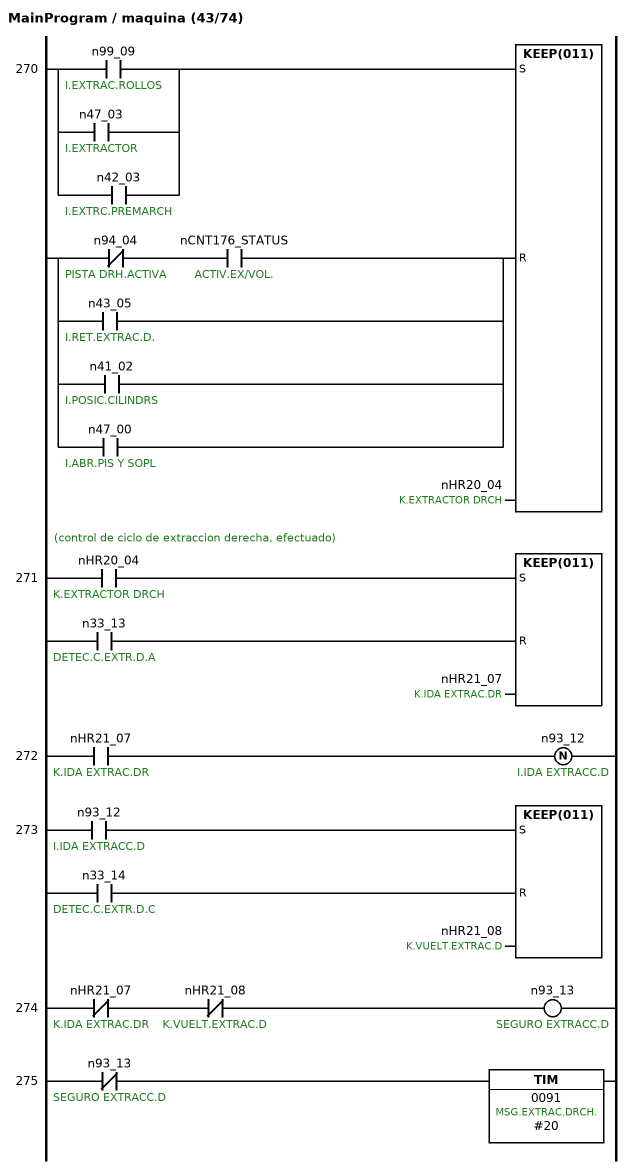
; [picture p48: MainProgram / maquina, rungs 270-275]
; rung 270
LD n99_09  ; I.EXTRAC.ROLLOS
OR n47_03  ; I.EXTRACTOR
OR n42_03  ; I.EXTRC.PREMARCH
LDNOT n94_04  ; PISTA DRH.ACTIVA
AND nCNT176_STATUS  ; ACTIV.EX/VOL.
OR n43_05  ; I.RET.EXTRAC.D.
OR n41_02  ; I.POSIC.CILINDRS
OR n47_00  ; I.ABR.PIS Y SOPL
KEEP(011) nHR20_04  ; K.EXTRACTOR DRCH
; rung 271: (control de ciclo de extraccion derecha, efectuado)
LD nHR20_04  ; K.EXTRACTOR DRCH
LD n33_13  ; DETEC.C.EXTR.D.A
KEEP(011) nHR21_07  ; K.IDA EXTRAC.DR
; rung 272
LD nHR21_07  ; K.IDA EXTRAC.DR
DIFD(014) n93_12  ; I.IDA EXTRACC.D
; rung 273
LD n93_12  ; I.IDA EXTRACC.D
LD n33_14  ; DETEC.C.EXTR.D.C
KEEP(011) nHR21_08  ; K.VUELT.EXTRAC.D
; rung 274
LDNOT nHR21_07  ; K.IDA EXTRAC.DR
ANDNOT nHR21_08  ; K.VUELT.EXTRAC.D
OUT n93_13  ; SEGURO EXTRACC.D
; rung 275
LDNOT n93_13  ; SEGURO EXTRACC.D
TIM 0091 #20  ; MSG.EXTRAC.DRCH.

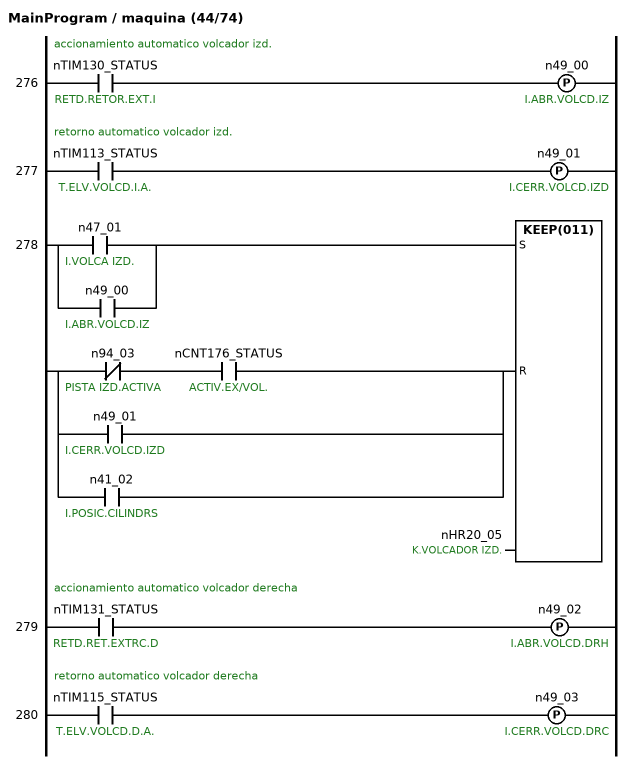
; rung 276: accionamiento automatico volcador izd.
LD nTIM130_STATUS  ; RETD.RETOR.EXT.I
DIFU(013) n49_00  ; I.ABR.VOLCD.IZ
; rung 277: retorno automatico volcador izd.
LD nTIM113_STATUS  ; T.ELV.VOLCD.I.A.
DIFU(013) n49_01  ; I.CERR.VOLCD.IZD
; rung 278
LD n47_01  ; I.VOLCA IZD.
OR n49_00  ; I.ABR.VOLCD.IZ
LDNOT n94_03  ; PISTA IZD.ACTIVA
AND nCNT176_STATUS  ; ACTIV.EX/VOL.
OR n49_01  ; I.CERR.VOLCD.IZD
OR n41_02  ; I.POSIC.CILINDRS
KEEP(011) nHR20_05  ; K.VOLCADOR IZD.
; rung 279: accionamiento automatico volcador derecha
LD nTIM131_STATUS  ; RETD.RET.EXTRC.D
DIFU(013) n49_02  ; I.ABR.VOLCD.DRH
; rung 280: retorno automatico volcador derecha
LD nTIM115_STATUS  ; T.ELV.VOLCD.D.A.
DIFU(013) n49_03  ; I.CERR.VOLCD.DRC

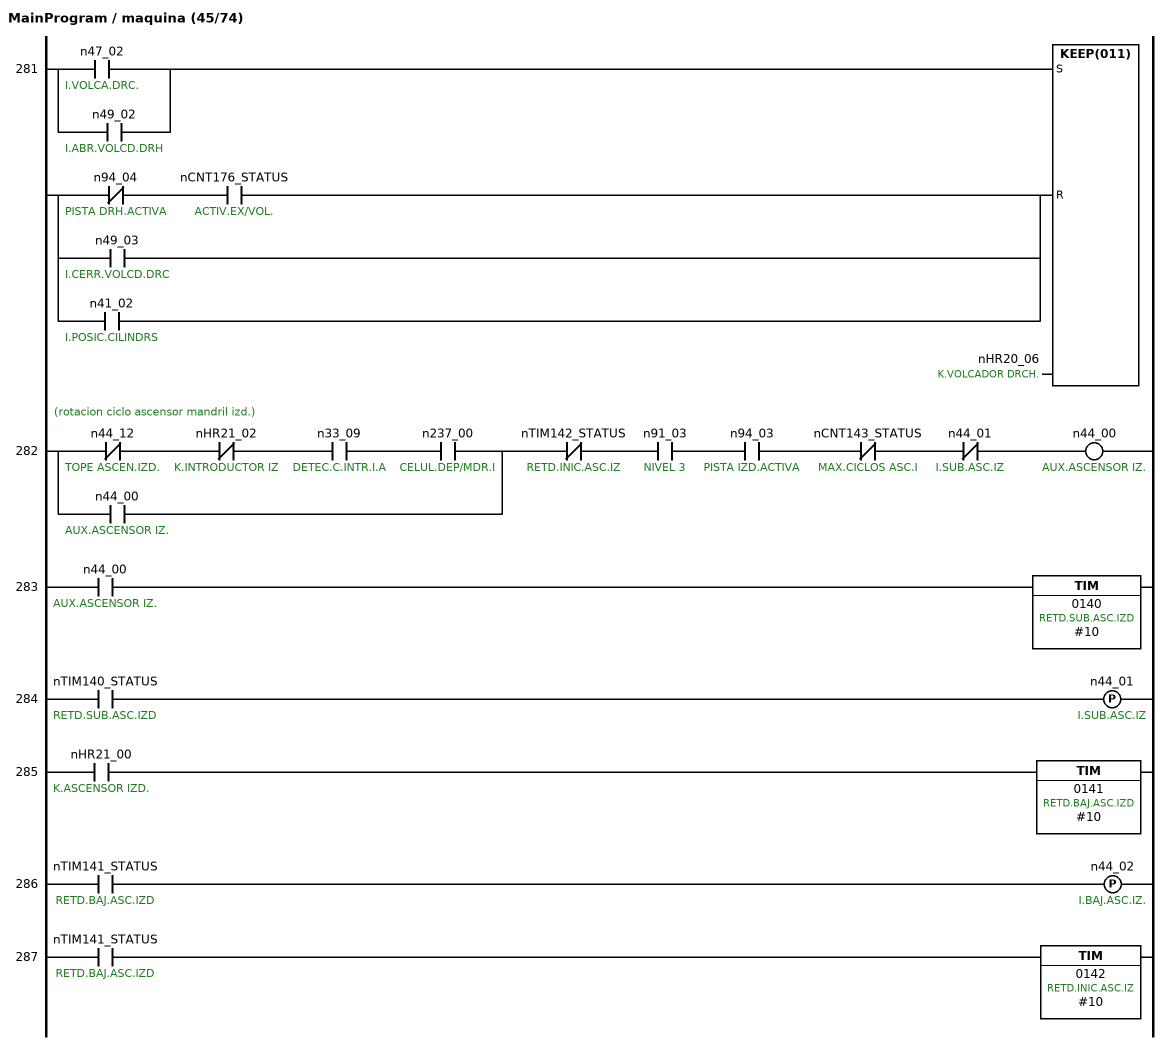
; rung 281
LD n47_02  ; I.VOLCA.DRC.
OR n49_02  ; I.ABR.VOLCD.DRH
LDNOT n94_04  ; PISTA DRH.ACTIVA
AND nCNT176_STATUS  ; ACTIV.EX/VOL.
OR n49_03  ; I.CERR.VOLCD.DRC
OR n41_02  ; I.POSIC.CILINDRS
KEEP(011) nHR20_06  ; K.VOLCADOR DRCH.
; rung 282: (rotacion ciclo ascensor mandril izd.)
LDNOT n44_12  ; TOPE ASCEN.IZD.
ANDNOT nHR21_02  ; K.INTRODUCTOR IZ
AND n33_09  ; DETEC.C.INTR.I.A
AND n237_00  ; CELUL.DEP/MDR.I
OR n44_00  ; AUX.ASCENSOR IZ.
ANDNOT nTIM142_STATUS  ; RETD.INIC.ASC.IZ
AND n91_03  ; NIVEL 3
AND n94_03  ; PISTA IZD.ACTIVA
ANDNOT nCNT143_STATUS  ; MAX.CICLOS ASC.I
ANDNOT n44_01  ; I.SUB.ASC.IZ
OUT n44_00  ; AUX.ASCENSOR IZ.
; rung 283
LD n44_00  ; AUX.ASCENSOR IZ.
TIM 0140 #10  ; RETD.SUB.ASC.IZD
; rung 284
LD nTIM140_STATUS  ; RETD.SUB.ASC.IZD
DIFU(013) n44_01  ; I.SUB.ASC.IZ
; rung 285
LD nHR21_00  ; K.ASCENSOR IZD.
TIM 0141 #10  ; RETD.BAJ.ASC.IZD
; rung 286
LD nTIM141_STATUS  ; RETD.BAJ.ASC.IZD
DIFU(013) n44_02  ; I.BAJ.ASC.IZ.
; rung 287
LD nTIM141_STATUS  ; RETD.BAJ.ASC.IZD
TIM 0142 #10  ; RETD.INIC.ASC.IZ

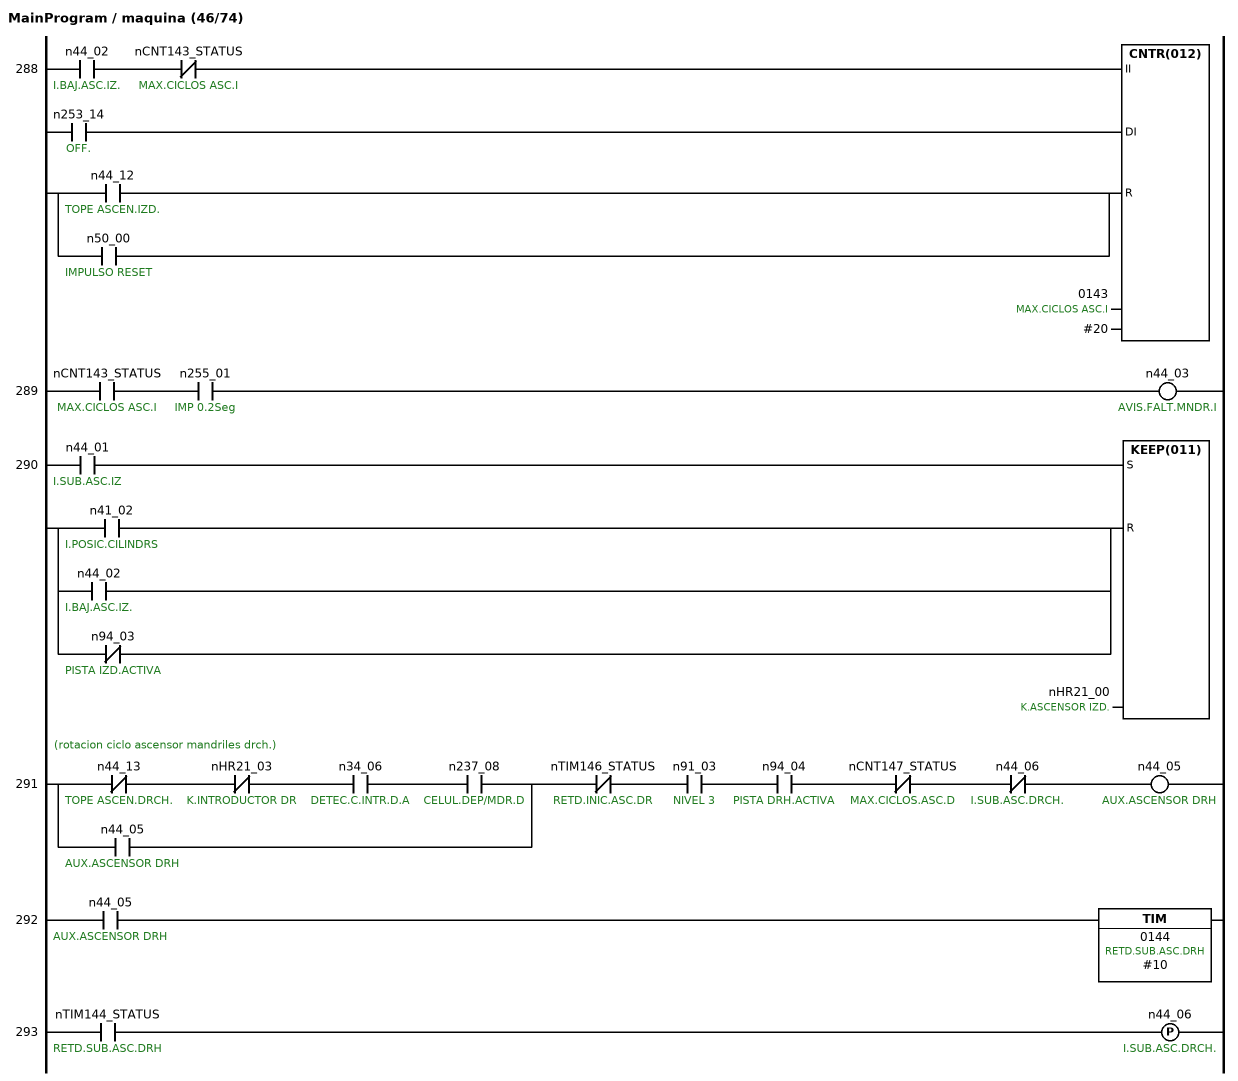
; rung 288
LD n44_02  ; I.BAJ.ASC.IZ.
ANDNOT nCNT143_STATUS  ; MAX.CICLOS ASC.I
LD n253_14  ; OFF.
LD n44_12  ; TOPE ASCEN.IZD.
OR n50_00  ; IMPULSO RESET
CNTR(012) 0143 #20  ; MAX.CICLOS ASC.I
; rung 289
LD nCNT143_STATUS  ; MAX.CICLOS ASC.I
AND n255_01  ; IMP 0.2Seg
OUT n44_03  ; AVIS.FALT.MNDR.I
; rung 290
LD n44_01  ; I.SUB.ASC.IZ
LD n41_02  ; I.POSIC.CILINDRS
OR n44_02  ; I.BAJ.ASC.IZ.
ORNOT n94_03  ; PISTA IZD.ACTIVA
KEEP(011) nHR21_00  ; K.ASCENSOR IZD.
; rung 291: (rotacion ciclo ascensor mandriles drch.)
LDNOT n44_13  ; TOPE ASCEN.DRCH.
ANDNOT nHR21_03  ; K.INTRODUCTOR DR
AND n34_06  ; DETEC.C.INTR.D.A
AND n237_08  ; CELUL.DEP/MDR.D
OR n44_05  ; AUX.ASCENSOR DRH
ANDNOT nTIM146_STATUS  ; RETD.INIC.ASC.DR
AND n91_03  ; NIVEL 3
AND n94_04  ; PISTA DRH.ACTIVA
ANDNOT nCNT147_STATUS  ; MAX.CICLOS.ASC.D
ANDNOT n44_06  ; I.SUB.ASC.DRCH.
OUT n44_05  ; AUX.ASCENSOR DRH
; rung 292
LD n44_05  ; AUX.ASCENSOR DRH
TIM 0144 #10  ; RETD.SUB.ASC.DRH
; rung 293
LD nTIM144_STATUS  ; RETD.SUB.ASC.DRH
DIFU(013) n44_06  ; I.SUB.ASC.DRCH.

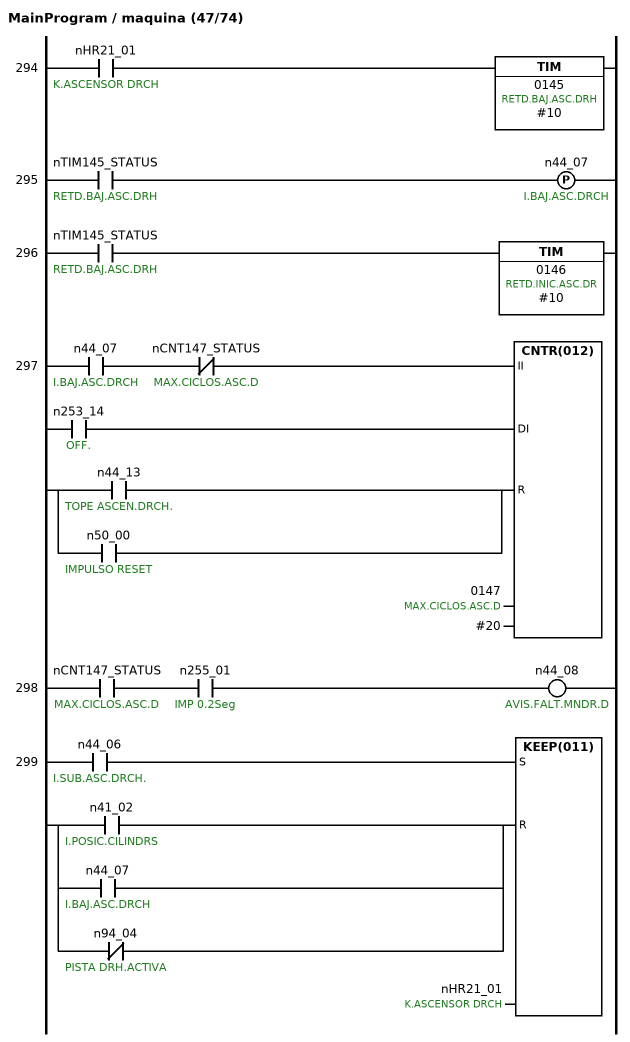
; rung 294
LD nHR21_01  ; K.ASCENSOR DRCH
TIM 0145 #10  ; RETD.BAJ.ASC.DRH
; rung 295
LD nTIM145_STATUS  ; RETD.BAJ.ASC.DRH
DIFU(013) n44_07  ; I.BAJ.ASC.DRCH
; rung 296
LD nTIM145_STATUS  ; RETD.BAJ.ASC.DRH
TIM 0146 #10  ; RETD.INIC.ASC.DR
; rung 297
LD n44_07  ; I.BAJ.ASC.DRCH
ANDNOT nCNT147_STATUS  ; MAX.CICLOS.ASC.D
LD n253_14  ; OFF.
LD n44_13  ; TOPE ASCEN.DRCH.
OR n50_00  ; IMPULSO RESET
CNTR(012) 0147 #20  ; MAX.CICLOS.ASC.D
; rung 298
LD nCNT147_STATUS  ; MAX.CICLOS.ASC.D
AND n255_01  ; IMP 0.2Seg
OUT n44_08  ; AVIS.FALT.MNDR.D
; rung 299
LD n44_06  ; I.SUB.ASC.DRCH.
LD n41_02  ; I.POSIC.CILINDRS
OR n44_07  ; I.BAJ.ASC.DRCH
ORNOT n94_04  ; PISTA DRH.ACTIVA
KEEP(011) nHR21_01  ; K.ASCENSOR DRCH

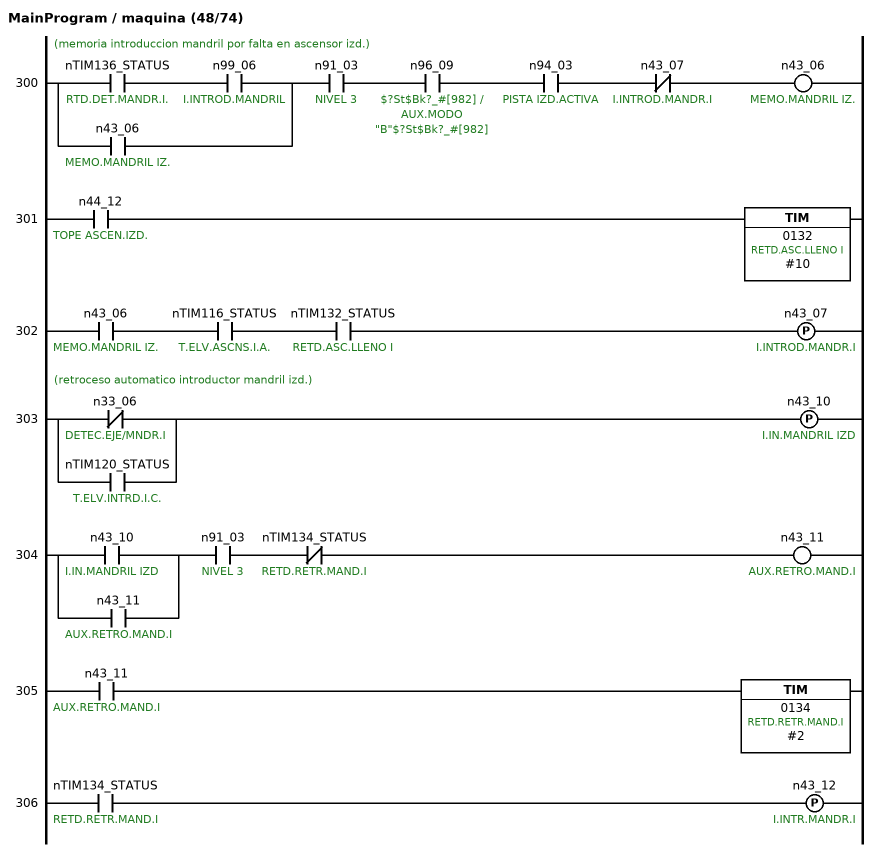
; rung 300: (memoria introduccion mandril por falta en ascensor izd.)
LD nTIM136_STATUS  ; RTD.DET.MANDR.I.
AND n99_06  ; I.INTROD.MANDRIL
OR n43_06  ; MEMO.MANDRIL IZ.
AND n91_03  ; NIVEL 3
AND n96_09  ; $?St$Bk?_#[982] / AUX.MODO "B"$?St$Bk?_#[982]
AND n94_03  ; PISTA IZD.ACTIVA
ANDNOT n43_07  ; I.INTROD.MANDR.I
OUT n43_06  ; MEMO.MANDRIL IZ.
; rung 301
LD n44_12  ; TOPE ASCEN.IZD.
TIM 0132 #10  ; RETD.ASC.LLENO I
; rung 302
LD n43_06  ; MEMO.MANDRIL IZ.
AND nTIM116_STATUS  ; T.ELV.ASCNS.I.A.
AND nTIM132_STATUS  ; RETD.ASC.LLENO I
DIFU(013) n43_07  ; I.INTROD.MANDR.I
; rung 303: (retroceso automatico introductor mandril izd.)
LDNOT n33_06  ; DETEC.EJE/MNDR.I
OR nTIM120_STATUS  ; T.ELV.INTRD.I.C.
DIFU(013) n43_10  ; I.IN.MANDRIL IZD
; rung 304
LD n43_10  ; I.IN.MANDRIL IZD
OR n43_11  ; AUX.RETRO.MAND.I
AND n91_03  ; NIVEL 3
ANDNOT nTIM134_STATUS  ; RETD.RETR.MAND.I
OUT n43_11  ; AUX.RETRO.MAND.I
; rung 305
LD n43_11  ; AUX.RETRO.MAND.I
TIM 0134 #2  ; RETD.RETR.MAND.I
; rung 306
LD nTIM134_STATUS  ; RETD.RETR.MAND.I
DIFU(013) n43_12  ; I.INTR.MANDR.I

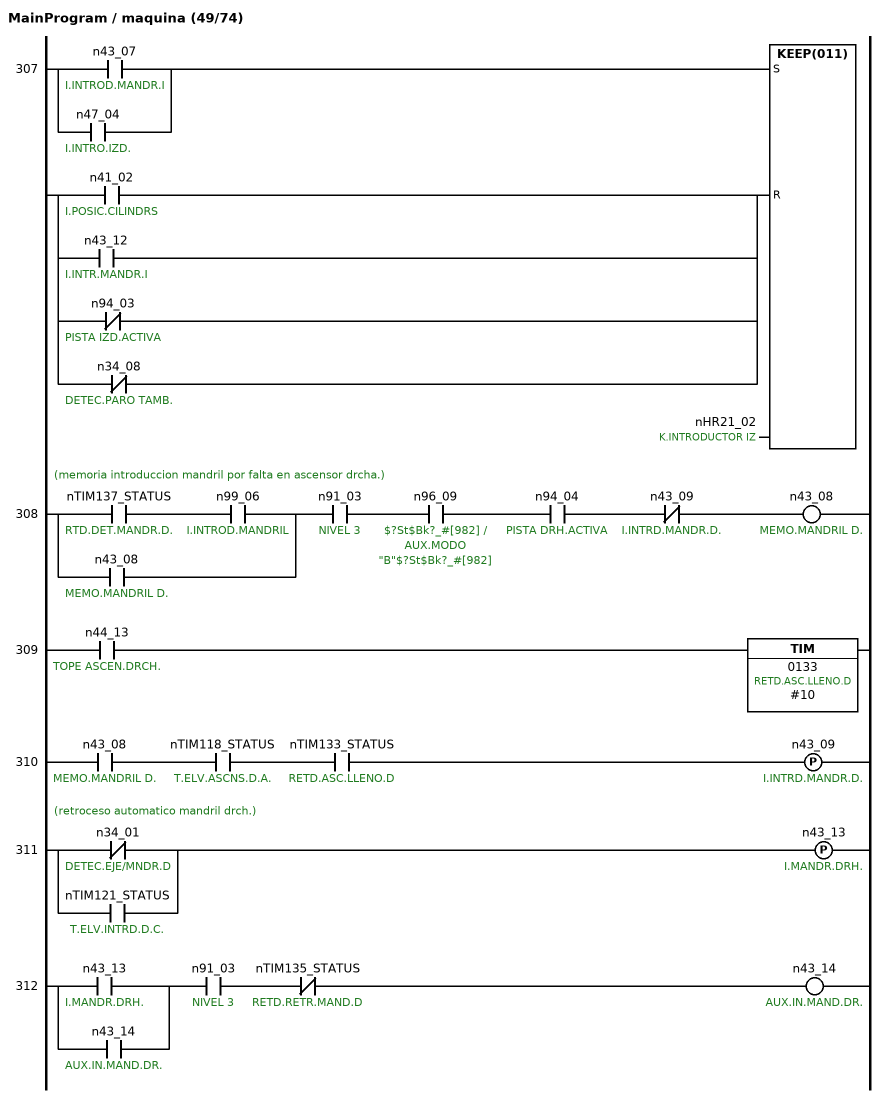
; rung 307
LD n43_07  ; I.INTROD.MANDR.I
OR n47_04  ; I.INTRO.IZD.
LD n41_02  ; I.POSIC.CILINDRS
OR n43_12  ; I.INTR.MANDR.I
ORNOT n94_03  ; PISTA IZD.ACTIVA
ORNOT n34_08  ; DETEC.PARO TAMB.
KEEP(011) nHR21_02  ; K.INTRODUCTOR IZ
; rung 308: (memoria introduccion mandril por falta en ascensor drcha.)
LD nTIM137_STATUS  ; RTD.DET.MANDR.D.
AND n99_06  ; I.INTROD.MANDRIL
OR n43_08  ; MEMO.MANDRIL D.
AND n91_03  ; NIVEL 3
AND n96_09  ; $?St$Bk?_#[982] / AUX.MODO "B"$?St$Bk?_#[982]
AND n94_04  ; PISTA DRH.ACTIVA
ANDNOT n43_09  ; I.INTRD.MANDR.D.
OUT n43_08  ; MEMO.MANDRIL D.
; rung 309
LD n44_13  ; TOPE ASCEN.DRCH.
TIM 0133 #10  ; RETD.ASC.LLENO.D
; rung 310
LD n43_08  ; MEMO.MANDRIL D.
AND nTIM118_STATUS  ; T.ELV.ASCNS.D.A.
AND nTIM133_STATUS  ; RETD.ASC.LLENO.D
DIFU(013) n43_09  ; I.INTRD.MANDR.D.
; rung 311: (retroceso automatico mandril drch.)
LDNOT n34_01  ; DETEC.EJE/MNDR.D
OR nTIM121_STATUS  ; T.ELV.INTRD.D.C.
DIFU(013) n43_13  ; I.MANDR.DRH.
; rung 312
LD n43_13  ; I.MANDR.DRH.
OR n43_14  ; AUX.IN.MAND.DR.
AND n91_03  ; NIVEL 3
ANDNOT nTIM135_STATUS  ; RETD.RETR.MAND.D
OUT n43_14  ; AUX.IN.MAND.DR.

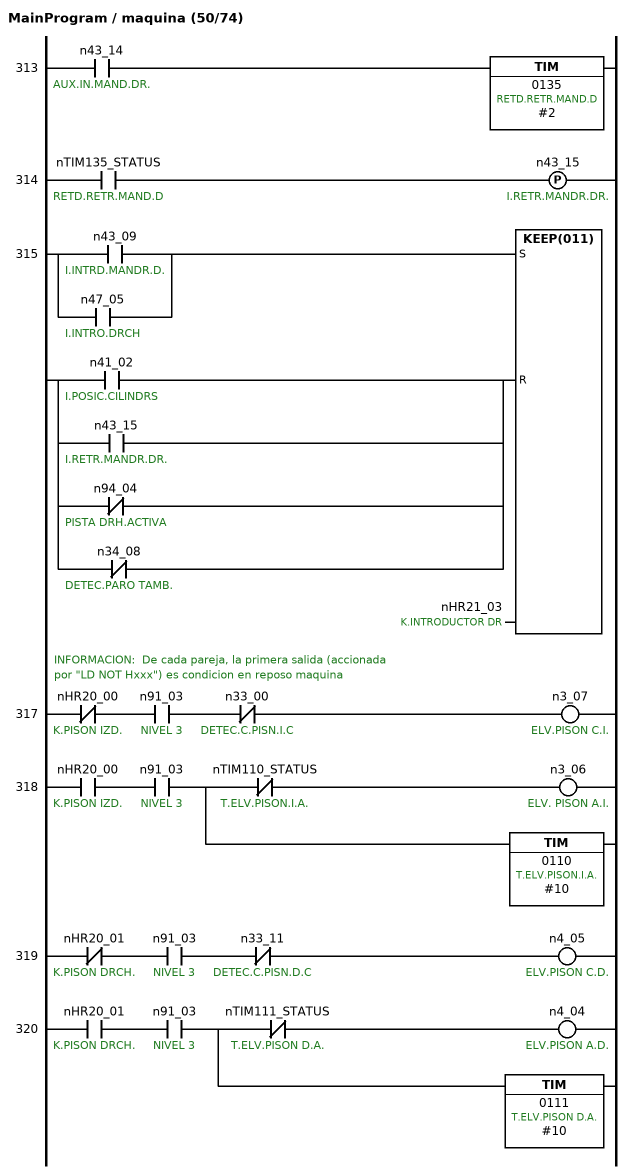
; rung 313
LD n43_14  ; AUX.IN.MAND.DR.
TIM 0135 #2  ; RETD.RETR.MAND.D
; rung 314
LD nTIM135_STATUS  ; RETD.RETR.MAND.D
DIFU(013) n43_15  ; I.RETR.MANDR.DR.
; rung 315
LD n43_09  ; I.INTRD.MANDR.D.
OR n47_05  ; I.INTRO.DRCH
LD n41_02  ; I.POSIC.CILINDRS
OR n43_15  ; I.RETR.MANDR.DR.
ORNOT n94_04  ; PISTA DRH.ACTIVA
ORNOT n34_08  ; DETEC.PARO TAMB.
KEEP(011) nHR21_03  ; K.INTRODUCTOR DR
; rung 316: ACCIONAMIENTO ELVS. REBOBINADOR, VOLCADORES Y CARGADORES / ------------------------------------------------------------
; rung 317: INFORMACION:  De cada pareja, la primera salida (accionada / por "LD NOT Hxxx") es condicion en reposo maquina
LDNOT nHR20_00  ; K.PISON IZD.
AND n91_03  ; NIVEL 3
ANDNOT n33_00  ; DETEC.C.PISN.I.C
OUT n3_07  ; ELV.PISON C.I.
; rung 318
LD nHR20_00  ; K.PISON IZD.
AND n91_03  ; NIVEL 3
OUT TR0
ANDNOT nTIM110_STATUS  ; T.ELV.PISON.I.A.
OUT n3_06  ; ELV. PISON A.I.
LD TR0
TIM 0110 #10  ; T.ELV.PISON.I.A.
; rung 319
LDNOT nHR20_01  ; K.PISON DRCH.
AND n91_03  ; NIVEL 3
ANDNOT n33_11  ; DETEC.C.PISN.D.C
OUT n4_05  ; ELV.PISON C.D.
; rung 320
LD nHR20_01  ; K.PISON DRCH.
AND n91_03  ; NIVEL 3
OUT TR0
ANDNOT nTIM111_STATUS  ; T.ELV.PISON D.A.
OUT n4_04  ; ELV.PISON A.D.
LD TR0
TIM 0111 #10  ; T.ELV.PISON D.A.

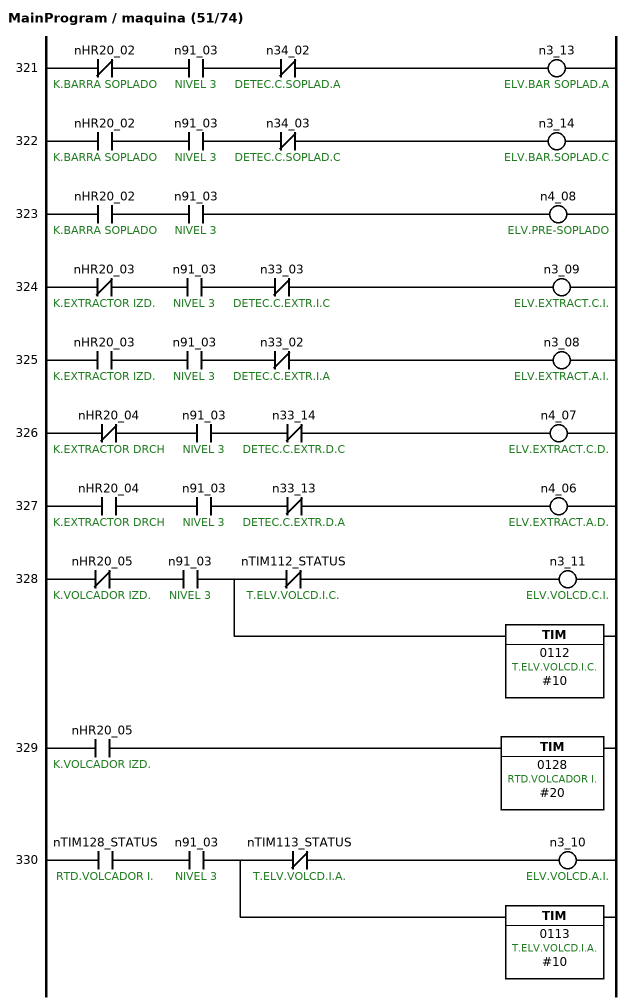
; rung 321
LDNOT nHR20_02  ; K.BARRA SOPLADO
AND n91_03  ; NIVEL 3
ANDNOT n34_02  ; DETEC.C.SOPLAD.A
OUT n3_13  ; ELV.BAR SOPLAD.A
; rung 322
LD nHR20_02  ; K.BARRA SOPLADO
AND n91_03  ; NIVEL 3
ANDNOT n34_03  ; DETEC.C.SOPLAD.C
OUT n3_14  ; ELV.BAR.SOPLAD.C
; rung 323
LD nHR20_02  ; K.BARRA SOPLADO
AND n91_03  ; NIVEL 3
OUT n4_08  ; ELV.PRE-SOPLADO
; rung 324
LDNOT nHR20_03  ; K.EXTRACTOR IZD.
AND n91_03  ; NIVEL 3
ANDNOT n33_03  ; DETEC.C.EXTR.I.C
OUT n3_09  ; ELV.EXTRACT.C.I.
; rung 325
LD nHR20_03  ; K.EXTRACTOR IZD.
AND n91_03  ; NIVEL 3
ANDNOT n33_02  ; DETEC.C.EXTR.I.A
OUT n3_08  ; ELV.EXTRACT.A.I.
; rung 326
LDNOT nHR20_04  ; K.EXTRACTOR DRCH
AND n91_03  ; NIVEL 3
ANDNOT n33_14  ; DETEC.C.EXTR.D.C
OUT n4_07  ; ELV.EXTRACT.C.D.
; rung 327
LD nHR20_04  ; K.EXTRACTOR DRCH
AND n91_03  ; NIVEL 3
ANDNOT n33_13  ; DETEC.C.EXTR.D.A
OUT n4_06  ; ELV.EXTRACT.A.D.
; rung 328
LDNOT nHR20_05  ; K.VOLCADOR IZD.
AND n91_03  ; NIVEL 3
OUT TR0
ANDNOT nTIM112_STATUS  ; T.ELV.VOLCD.I.C.
OUT n3_11  ; ELV.VOLCD.C.I.
LD TR0
TIM 0112 #10  ; T.ELV.VOLCD.I.C.
; rung 329
LD nHR20_05  ; K.VOLCADOR IZD.
TIM 0128 #20  ; RTD.VOLCADOR I.
; rung 330
LD nTIM128_STATUS  ; RTD.VOLCADOR I.
AND n91_03  ; NIVEL 3
OUT TR0
ANDNOT nTIM113_STATUS  ; T.ELV.VOLCD.I.A.
OUT n3_10  ; ELV.VOLCD.A.I.
LD TR0
TIM 0113 #10  ; T.ELV.VOLCD.I.A.

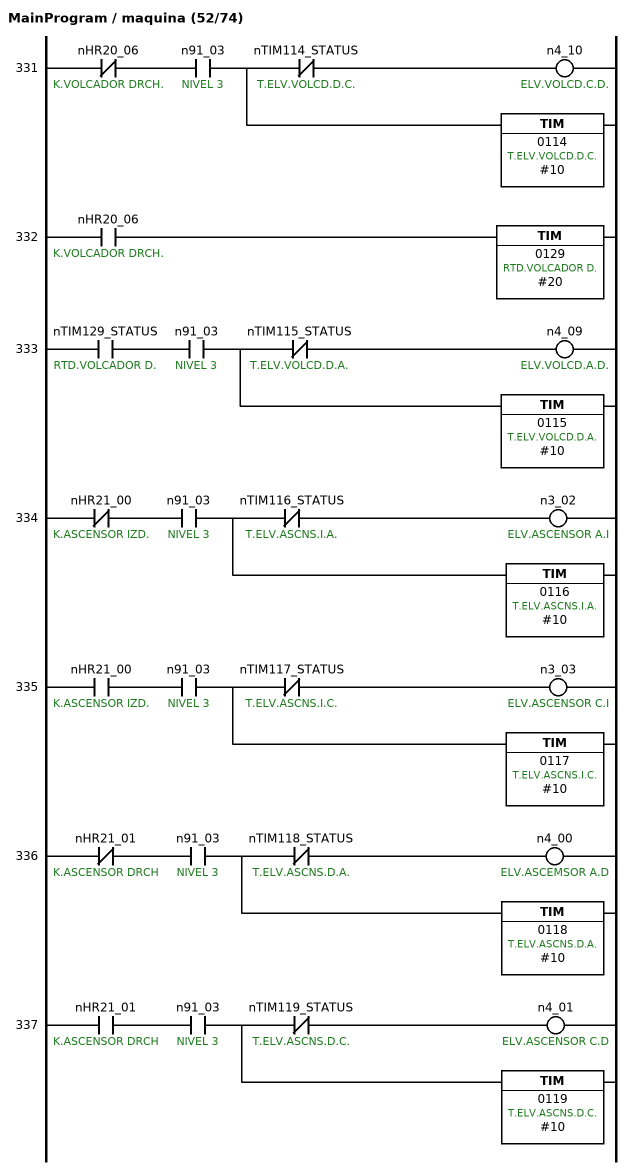
; rung 331
LDNOT nHR20_06  ; K.VOLCADOR DRCH.
AND n91_03  ; NIVEL 3
OUT TR0
ANDNOT nTIM114_STATUS  ; T.ELV.VOLCD.D.C.
OUT n4_10  ; ELV.VOLCD.C.D.
LD TR0
TIM 0114 #10  ; T.ELV.VOLCD.D.C.
; rung 332
LD nHR20_06  ; K.VOLCADOR DRCH.
TIM 0129 #20  ; RTD.VOLCADOR D.
; rung 333
LD nTIM129_STATUS  ; RTD.VOLCADOR D.
AND n91_03  ; NIVEL 3
OUT TR0
ANDNOT nTIM115_STATUS  ; T.ELV.VOLCD.D.A.
OUT n4_09  ; ELV.VOLCD.A.D.
LD TR0
TIM 0115 #10  ; T.ELV.VOLCD.D.A.
; rung 334
LDNOT nHR21_00  ; K.ASCENSOR IZD.
AND n91_03  ; NIVEL 3
OUT TR0
ANDNOT nTIM116_STATUS  ; T.ELV.ASCNS.I.A.
OUT n3_02  ; ELV.ASCENSOR A.I
LD TR0
TIM 0116 #10  ; T.ELV.ASCNS.I.A.
; rung 335
LD nHR21_00  ; K.ASCENSOR IZD.
AND n91_03  ; NIVEL 3
OUT TR0
ANDNOT nTIM117_STATUS  ; T.ELV.ASCNS.I.C.
OUT n3_03  ; ELV.ASCENSOR C.I
LD TR0
TIM 0117 #10  ; T.ELV.ASCNS.I.C.
; rung 336
LDNOT nHR21_01  ; K.ASCENSOR DRCH
AND n91_03  ; NIVEL 3
OUT TR0
ANDNOT nTIM118_STATUS  ; T.ELV.ASCNS.D.A.
OUT n4_00  ; ELV.ASCEMSOR A.D
LD TR0
TIM 0118 #10  ; T.ELV.ASCNS.D.A.
; rung 337
LD nHR21_01  ; K.ASCENSOR DRCH
AND n91_03  ; NIVEL 3
OUT TR0
ANDNOT nTIM119_STATUS  ; T.ELV.ASCNS.D.C.
OUT n4_01  ; ELV.ASCENSOR C.D
LD TR0
TIM 0119 #10  ; T.ELV.ASCNS.D.C.

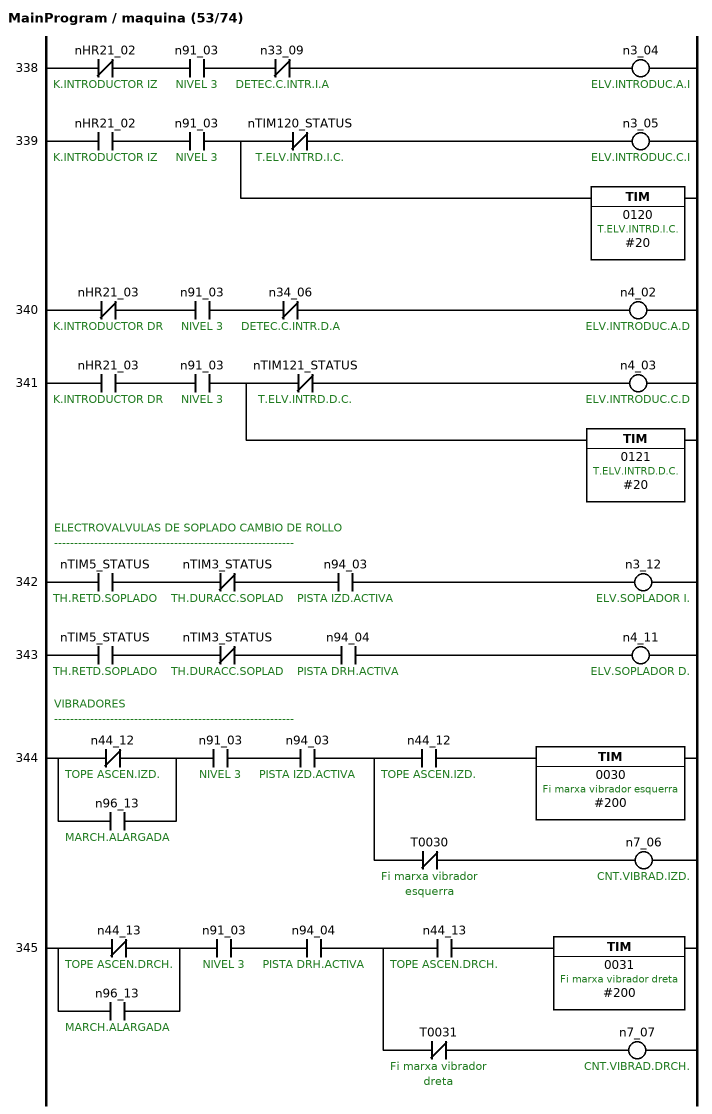
; rung 338
LDNOT nHR21_02  ; K.INTRODUCTOR IZ
AND n91_03  ; NIVEL 3
ANDNOT n33_09  ; DETEC.C.INTR.I.A
OUT n3_04  ; ELV.INTRODUC.A.I
; rung 339
LD nHR21_02  ; K.INTRODUCTOR IZ
AND n91_03  ; NIVEL 3
OUT TR0
ANDNOT nTIM120_STATUS  ; T.ELV.INTRD.I.C.
OUT n3_05  ; ELV.INTRODUC.C.I
LD TR0
TIM 0120 #20  ; T.ELV.INTRD.I.C.
; rung 340
LDNOT nHR21_03  ; K.INTRODUCTOR DR
AND n91_03  ; NIVEL 3
ANDNOT n34_06  ; DETEC.C.INTR.D.A
OUT n4_02  ; ELV.INTRODUC.A.D
; rung 341
LD nHR21_03  ; K.INTRODUCTOR DR
AND n91_03  ; NIVEL 3
OUT TR0
ANDNOT nTIM121_STATUS  ; T.ELV.INTRD.D.C.
OUT n4_03  ; ELV.INTRODUC.C.D
LD TR0
TIM 0121 #20  ; T.ELV.INTRD.D.C.
; rung 342: ELECTROVALVULAS DE SOPLADO CAMBIO DE ROLLO / ------------------------------------------------------------
LD nTIM5_STATUS  ; TH.RETD.SOPLADO
ANDNOT nTIM3_STATUS  ; TH.DURACC.SOPLAD
AND n94_03  ; PISTA IZD.ACTIVA
OUT n3_12  ; ELV.SOPLADOR I.
; rung 343
LD nTIM5_STATUS  ; TH.RETD.SOPLADO
ANDNOT nTIM3_STATUS  ; TH.DURACC.SOPLAD
AND n94_04  ; PISTA DRH.ACTIVA
OUT n4_11  ; ELV.SOPLADOR D.
; rung 344: VIBRADORES / ------------------------------------------------------------
LDNOT n44_12  ; TOPE ASCEN.IZD.
OR n96_13  ; MARCH.ALARGADA
AND n91_03  ; NIVEL 3
AND n94_03  ; PISTA IZD.ACTIVA
OUT TR0
AND n44_12  ; TOPE ASCEN.IZD.
TIM 0030 #200  ; Fi marxa vibrador esquerra
LD TR0
ANDNOT T0030  ; Fi marxa vibrador esquerra
OUT n7_06  ; CNT.VIBRAD.IZD.
; rung 345
LDNOT n44_13  ; TOPE ASCEN.DRCH.
OR n96_13  ; MARCH.ALARGADA
AND n91_03  ; NIVEL 3
AND n94_04  ; PISTA DRH.ACTIVA
OUT TR0
AND n44_13  ; TOPE ASCEN.DRCH.
TIM 0031 #200  ; Fi marxa vibrador dreta
LD TR0
ANDNOT T0031  ; Fi marxa vibrador dreta
OUT n7_07  ; CNT.VIBRAD.DRCH.

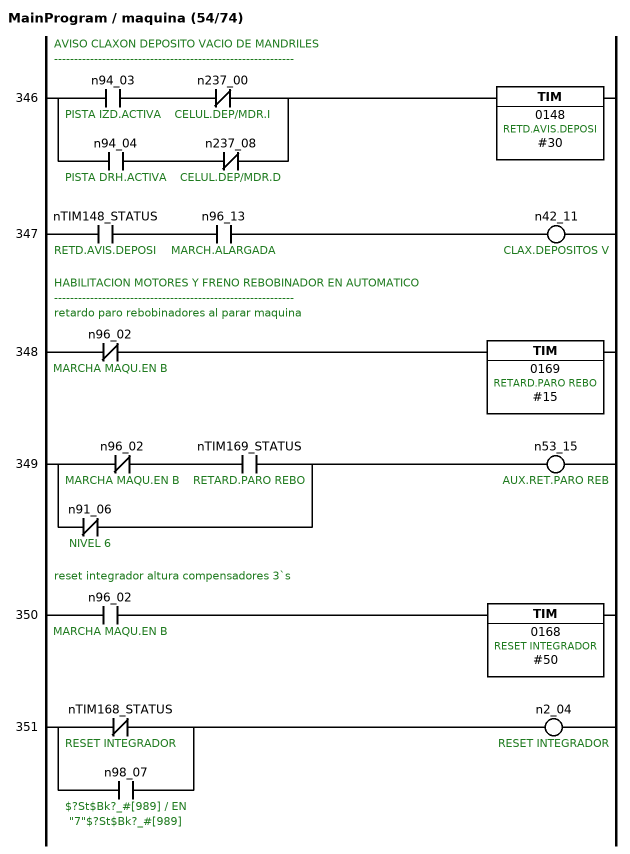
; rung 346: AVISO CLAXON DEPOSITO VACIO DE MANDRILES / ------------------------------------------------------------
LD n94_03  ; PISTA IZD.ACTIVA
ANDNOT n237_00  ; CELUL.DEP/MDR.I
LD n94_04  ; PISTA DRH.ACTIVA
ANDNOT n237_08  ; CELUL.DEP/MDR.D
ORLD
TIM 0148 #30  ; RETD.AVIS.DEPOSI
; rung 347
LD nTIM148_STATUS  ; RETD.AVIS.DEPOSI
AND n96_13  ; MARCH.ALARGADA
OUT n42_11  ; CLAX.DEPOSITOS V
; rung 348: HABILITACION MOTORES Y FRENO REBOBINADOR EN AUTOMATICO / ------------------------------------------------------------ / retardo paro rebobinadores al parar maquina
LDNOT n96_02  ; MARCHA MAQU.EN B
TIM 0169 #15  ; RETARD.PARO REBO
; rung 349
LDNOT n96_02  ; MARCHA MAQU.EN B
AND nTIM169_STATUS  ; RETARD.PARO REBO
ORNOT n91_06  ; NIVEL 6
OUT n53_15  ; AUX.RET.PARO REB
; rung 350: reset integrador altura compensadores 3`s
LD n96_02  ; MARCHA MAQU.EN B
TIM 0168 #50  ; RESET INTEGRADOR
; rung 351
LDNOT nTIM168_STATUS  ; RESET INTEGRADOR
OR n98_07  ; $?St$Bk?_#[989] / EN "7"$?St$Bk?_#[989]
OUT n2_04  ; RESET INTEGRADOR

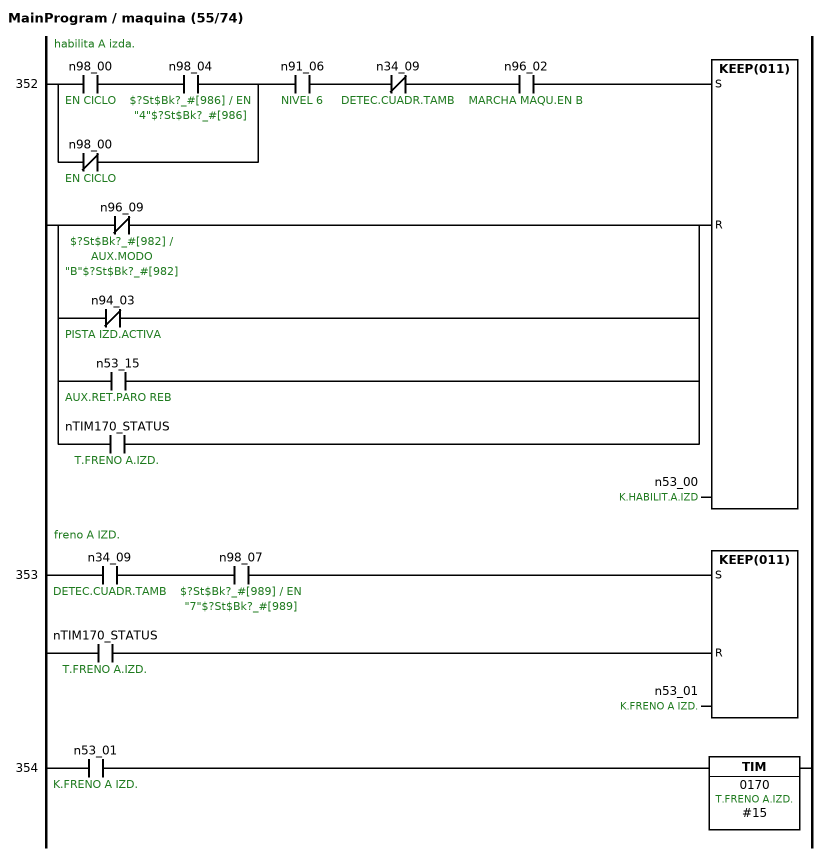
; rung 352: habilita A izda.
LD n98_00  ; EN CICLO
AND n98_04  ; $?St$Bk?_#[986] / EN "4"$?St$Bk?_#[986]
ORNOT n98_00  ; EN CICLO
AND n91_06  ; NIVEL 6
ANDNOT n34_09  ; DETEC.CUADR.TAMB
AND n96_02  ; MARCHA MAQU.EN B
LDNOT n96_09  ; $?St$Bk?_#[982] / AUX.MODO "B"$?St$Bk?_#[982]
ORNOT n94_03  ; PISTA IZD.ACTIVA
OR n53_15  ; AUX.RET.PARO REB
OR nTIM170_STATUS  ; T.FRENO A.IZD.
KEEP(011) n53_00  ; K.HABILIT.A.IZD
; rung 353: freno A IZD.
LD n34_09  ; DETEC.CUADR.TAMB
AND n98_07  ; $?St$Bk?_#[989] / EN "7"$?St$Bk?_#[989]
LD nTIM170_STATUS  ; T.FRENO A.IZD.
KEEP(011) n53_01  ; K.FRENO A IZD.
; rung 354
LD n53_01  ; K.FRENO A IZD.
TIM 0170 #15  ; T.FRENO A.IZD.

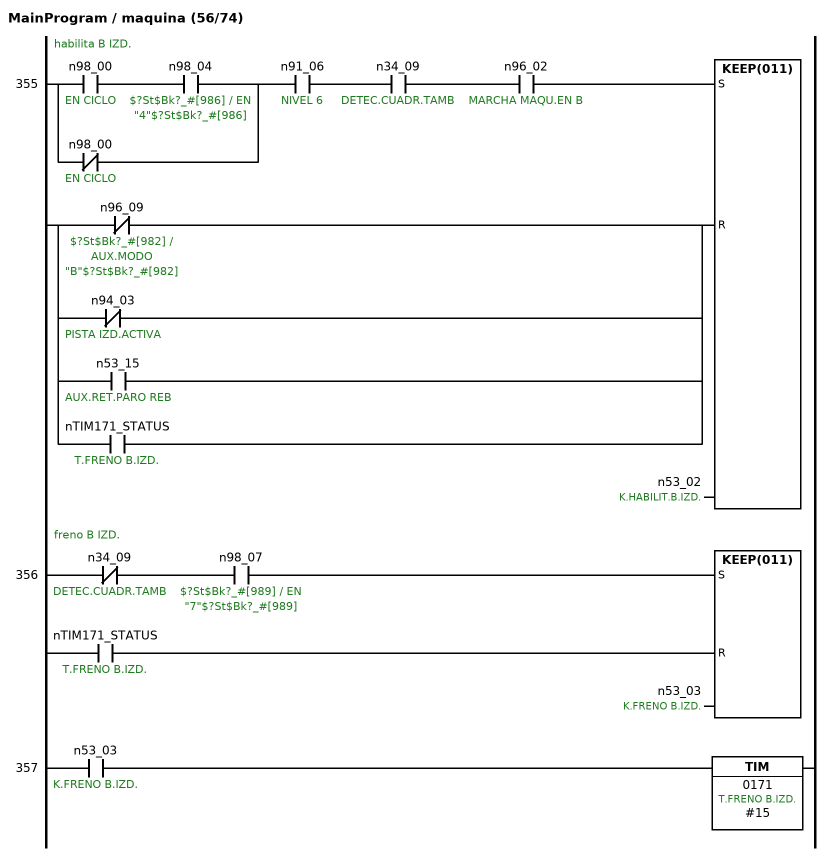
; rung 355: habilita B IZD.
LD n98_00  ; EN CICLO
AND n98_04  ; $?St$Bk?_#[986] / EN "4"$?St$Bk?_#[986]
ORNOT n98_00  ; EN CICLO
AND n91_06  ; NIVEL 6
AND n34_09  ; DETEC.CUADR.TAMB
AND n96_02  ; MARCHA MAQU.EN B
LDNOT n96_09  ; $?St$Bk?_#[982] / AUX.MODO "B"$?St$Bk?_#[982]
ORNOT n94_03  ; PISTA IZD.ACTIVA
OR n53_15  ; AUX.RET.PARO REB
OR nTIM171_STATUS  ; T.FRENO B.IZD.
KEEP(011) n53_02  ; K.HABILIT.B.IZD.
; rung 356: freno B IZD.
LDNOT n34_09  ; DETEC.CUADR.TAMB
AND n98_07  ; $?St$Bk?_#[989] / EN "7"$?St$Bk?_#[989]
LD nTIM171_STATUS  ; T.FRENO B.IZD.
KEEP(011) n53_03  ; K.FRENO B.IZD.
; rung 357
LD n53_03  ; K.FRENO B.IZD.
TIM 0171 #15  ; T.FRENO B.IZD.

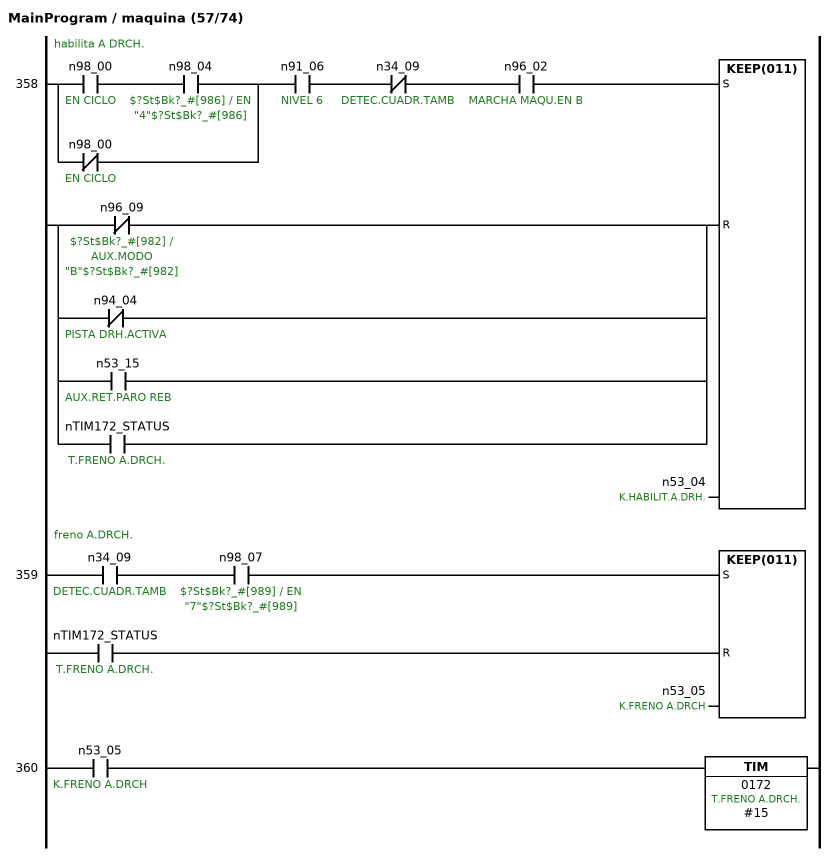
; rung 358: habilita A DRCH.
LD n98_00  ; EN CICLO
AND n98_04  ; $?St$Bk?_#[986] / EN "4"$?St$Bk?_#[986]
ORNOT n98_00  ; EN CICLO
AND n91_06  ; NIVEL 6
ANDNOT n34_09  ; DETEC.CUADR.TAMB
AND n96_02  ; MARCHA MAQU.EN B
LDNOT n96_09  ; $?St$Bk?_#[982] / AUX.MODO "B"$?St$Bk?_#[982]
ORNOT n94_04  ; PISTA DRH.ACTIVA
OR n53_15  ; AUX.RET.PARO REB
OR nTIM172_STATUS  ; T.FRENO A.DRCH.
KEEP(011) n53_04  ; K.HABILIT.A.DRH.
; rung 359: freno A.DRCH.
LD n34_09  ; DETEC.CUADR.TAMB
AND n98_07  ; $?St$Bk?_#[989] / EN "7"$?St$Bk?_#[989]
LD nTIM172_STATUS  ; T.FRENO A.DRCH.
KEEP(011) n53_05  ; K.FRENO A.DRCH
; rung 360
LD n53_05  ; K.FRENO A.DRCH
TIM 0172 #15  ; T.FRENO A.DRCH.

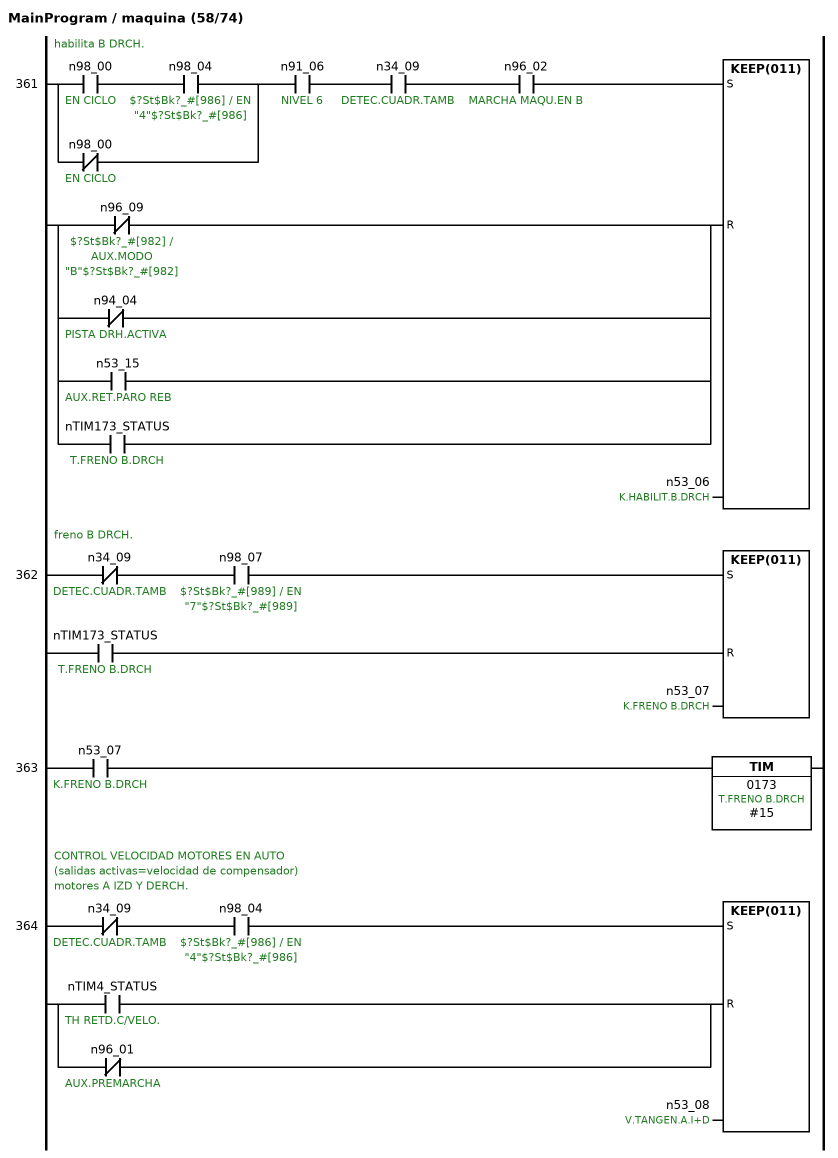
; rung 361: habilita B DRCH.
LD n98_00  ; EN CICLO
AND n98_04  ; $?St$Bk?_#[986] / EN "4"$?St$Bk?_#[986]
ORNOT n98_00  ; EN CICLO
AND n91_06  ; NIVEL 6
AND n34_09  ; DETEC.CUADR.TAMB
AND n96_02  ; MARCHA MAQU.EN B
LDNOT n96_09  ; $?St$Bk?_#[982] / AUX.MODO "B"$?St$Bk?_#[982]
ORNOT n94_04  ; PISTA DRH.ACTIVA
OR n53_15  ; AUX.RET.PARO REB
OR nTIM173_STATUS  ; T.FRENO B.DRCH
KEEP(011) n53_06  ; K.HABILIT.B.DRCH
; rung 362: freno B DRCH.
LDNOT n34_09  ; DETEC.CUADR.TAMB
AND n98_07  ; $?St$Bk?_#[989] / EN "7"$?St$Bk?_#[989]
LD nTIM173_STATUS  ; T.FRENO B.DRCH
KEEP(011) n53_07  ; K.FRENO B.DRCH
; rung 363
LD n53_07  ; K.FRENO B.DRCH
TIM 0173 #15  ; T.FRENO B.DRCH
; rung 364: CONTROL VELOCIDAD MOTORES EN AUTO / (salidas activas=velocidad de compensador) / motores A IZD Y DERCH.
LDNOT n34_09  ; DETEC.CUADR.TAMB
AND n98_04  ; $?St$Bk?_#[986] / EN "4"$?St$Bk?_#[986]
LD nTIM4_STATUS  ; TH RETD.C/VELO.
ORNOT n96_01  ; AUX.PREMARCHA
KEEP(011) n53_08  ; V.TANGEN.A.I+D

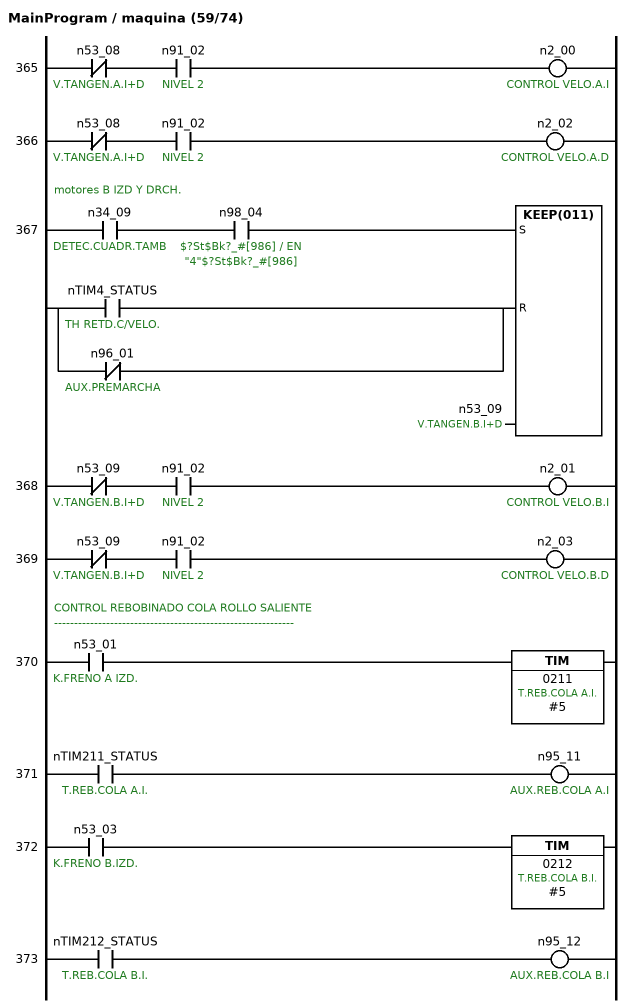
; rung 365
LDNOT n53_08  ; V.TANGEN.A.I+D
AND n91_02  ; NIVEL 2
OUT n2_00  ; CONTROL VELO.A.I
; rung 366
LDNOT n53_08  ; V.TANGEN.A.I+D
AND n91_02  ; NIVEL 2
OUT n2_02  ; CONTROL VELO.A.D
; rung 367: motores B IZD Y DRCH.
LD n34_09  ; DETEC.CUADR.TAMB
AND n98_04  ; $?St$Bk?_#[986] / EN "4"$?St$Bk?_#[986]
LD nTIM4_STATUS  ; TH RETD.C/VELO.
ORNOT n96_01  ; AUX.PREMARCHA
KEEP(011) n53_09  ; V.TANGEN.B.I+D
; rung 368
LDNOT n53_09  ; V.TANGEN.B.I+D
AND n91_02  ; NIVEL 2
OUT n2_01  ; CONTROL VELO.B.I
; rung 369
LDNOT n53_09  ; V.TANGEN.B.I+D
AND n91_02  ; NIVEL 2
OUT n2_03  ; CONTROL VELO.B.D
; rung 370: CONTROL REBOBINADO COLA ROLLO SALIENTE / ------------------------------------------------------------
LD n53_01  ; K.FRENO A IZD.
TIM 0211 #5  ; T.REB.COLA A.I.
; rung 371
LD nTIM211_STATUS  ; T.REB.COLA A.I.
OUT n95_11  ; AUX.REB.COLA A.I
; rung 372
LD n53_03  ; K.FRENO B.IZD.
TIM 0212 #5  ; T.REB.COLA B.I.
; rung 373
LD nTIM212_STATUS  ; T.REB.COLA B.I.
OUT n95_12  ; AUX.REB.COLA B.I

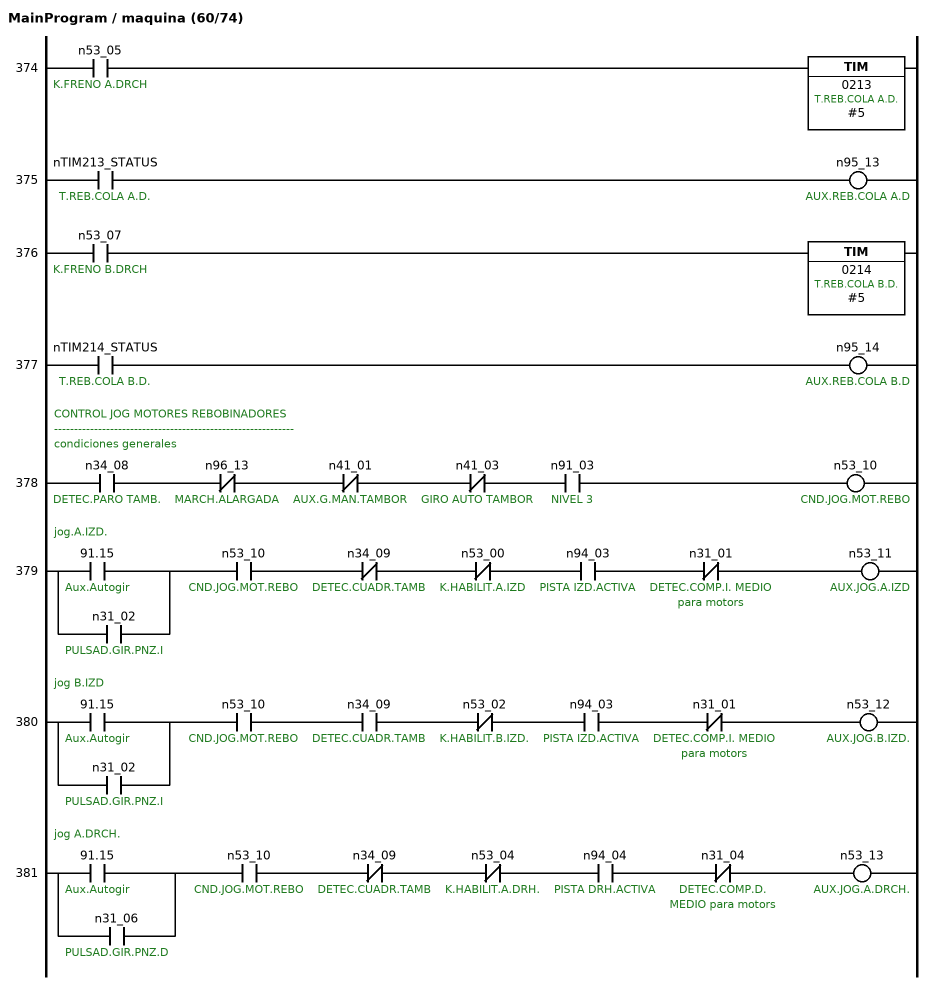
; rung 374
LD n53_05  ; K.FRENO A.DRCH
TIM 0213 #5  ; T.REB.COLA A.D.
; rung 375
LD nTIM213_STATUS  ; T.REB.COLA A.D.
OUT n95_13  ; AUX.REB.COLA A.D
; rung 376
LD n53_07  ; K.FRENO B.DRCH
TIM 0214 #5  ; T.REB.COLA B.D.
; rung 377
LD nTIM214_STATUS  ; T.REB.COLA B.D.
OUT n95_14  ; AUX.REB.COLA B.D
; rung 378: CONTROL JOG MOTORES REBOBINADORES / ------------------------------------------------------------ / condiciones generales
LD n34_08  ; DETEC.PARO TAMB.
ANDNOT n96_13  ; MARCH.ALARGADA
ANDNOT n41_01  ; AUX.G.MAN.TAMBOR
ANDNOT n41_03  ; GIRO AUTO TAMBOR
AND n91_03  ; NIVEL 3
OUT n53_10  ; CND.JOG.MOT.REBO
; rung 379: jog.A.IZD.
LD 91.15  ; Aux.Autogir
OR n31_02  ; PULSAD.GIR.PNZ.I
AND n53_10  ; CND.JOG.MOT.REBO
ANDNOT n34_09  ; DETEC.CUADR.TAMB
ANDNOT n53_00  ; K.HABILIT.A.IZD
AND n94_03  ; PISTA IZD.ACTIVA
ANDNOT n31_01  ; DETEC.COMP.I. MEDIO para motors
OUT n53_11  ; AUX.JOG.A.IZD
; rung 380: jog B.IZD
LD 91.15  ; Aux.Autogir
OR n31_02  ; PULSAD.GIR.PNZ.I
AND n53_10  ; CND.JOG.MOT.REBO
AND n34_09  ; DETEC.CUADR.TAMB
ANDNOT n53_02  ; K.HABILIT.B.IZD.
AND n94_03  ; PISTA IZD.ACTIVA
ANDNOT n31_01  ; DETEC.COMP.I. MEDIO para motors
OUT n53_12  ; AUX.JOG.B.IZD.
; rung 381: jog A.DRCH.
LD 91.15  ; Aux.Autogir
OR n31_06  ; PULSAD.GIR.PNZ.D
AND n53_10  ; CND.JOG.MOT.REBO
ANDNOT n34_09  ; DETEC.CUADR.TAMB
ANDNOT n53_04  ; K.HABILIT.A.DRH.
AND n94_04  ; PISTA DRH.ACTIVA
ANDNOT n31_04  ; DETEC.COMP.D. MEDIO para motors
OUT n53_13  ; AUX.JOG.A.DRCH.

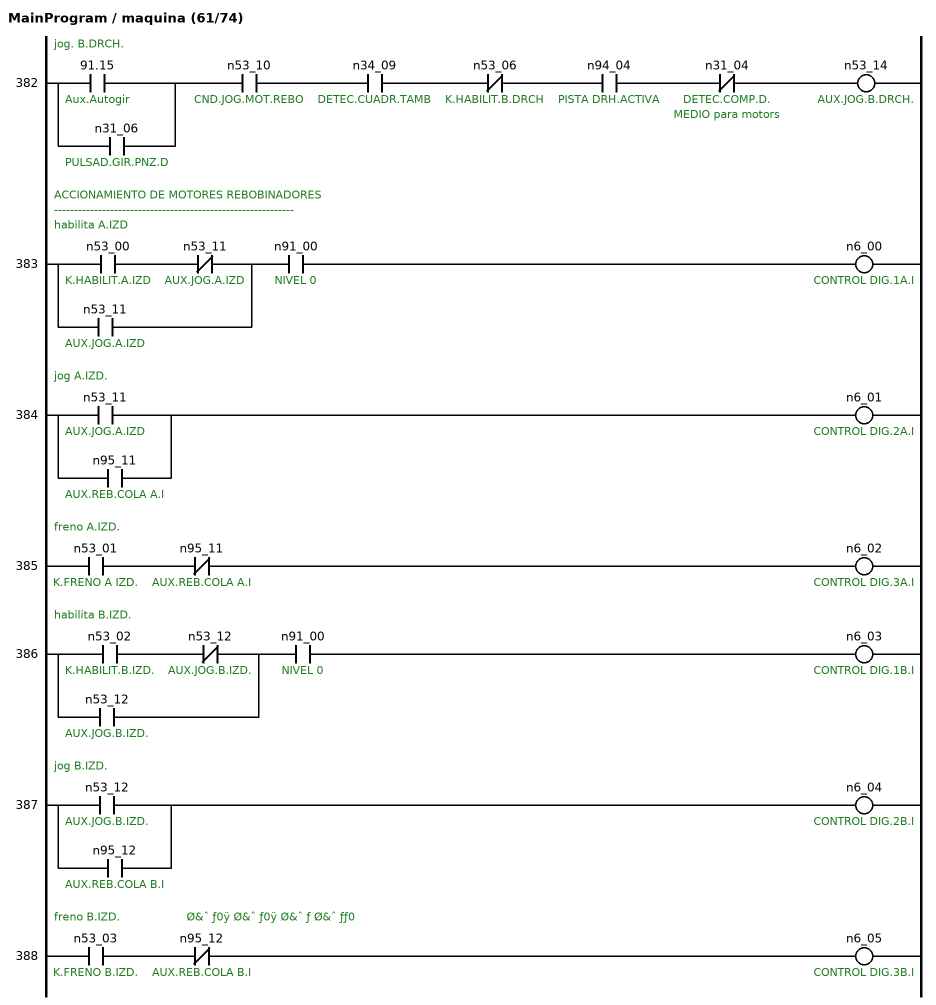
; rung 382: jog. B.DRCH.
LD 91.15  ; Aux.Autogir
OR n31_06  ; PULSAD.GIR.PNZ.D
AND n53_10  ; CND.JOG.MOT.REBO
AND n34_09  ; DETEC.CUADR.TAMB
ANDNOT n53_06  ; K.HABILIT.B.DRCH
AND n94_04  ; PISTA DRH.ACTIVA
ANDNOT n31_04  ; DETEC.COMP.D. MEDIO para motors
OUT n53_14  ; AUX.JOG.B.DRCH.
; rung 383: ACCIONAMIENTO DE MOTORES REBOBINADORES / ------------------------------------------------------------ / habilita A.IZD
LD n53_00  ; K.HABILIT.A.IZD
ANDNOT n53_11  ; AUX.JOG.A.IZD
OR n53_11  ; AUX.JOG.A.IZD
AND n91_00  ; NIVEL 0
OUT n6_00  ; CONTROL DIG.1A.I
; rung 384: jog A.IZD.
LD n53_11  ; AUX.JOG.A.IZD
OR n95_11  ; AUX.REB.COLA A.I
OUT n6_01  ; CONTROL DIG.2A.I
; rung 385: freno A.IZD.
LD n53_01  ; K.FRENO A IZD.
ANDNOT n95_11  ; AUX.REB.COLA A.I
OUT n6_02  ; CONTROL DIG.3A.I
; rung 386: habilita B.IZD.
LD n53_02  ; K.HABILIT.B.IZD.
ANDNOT n53_12  ; AUX.JOG.B.IZD.
OR n53_12  ; AUX.JOG.B.IZD.
AND n91_00  ; NIVEL 0
OUT n6_03  ; CONTROL DIG.1B.I
; rung 387: jog B.IZD.
LD n53_12  ; AUX.JOG.B.IZD.
OR n95_12  ; AUX.REB.COLA B.I
OUT n6_04  ; CONTROL DIG.2B.I
; rung 388: freno B.IZD.                   Ø&ˆƒ0ÿØ&ˆƒ0ÿØ&ˆƒØ&ˆƒƒ0
LD n53_03  ; K.FRENO B.IZD.
ANDNOT n95_12  ; AUX.REB.COLA B.I
OUT n6_05  ; CONTROL DIG.3B.I

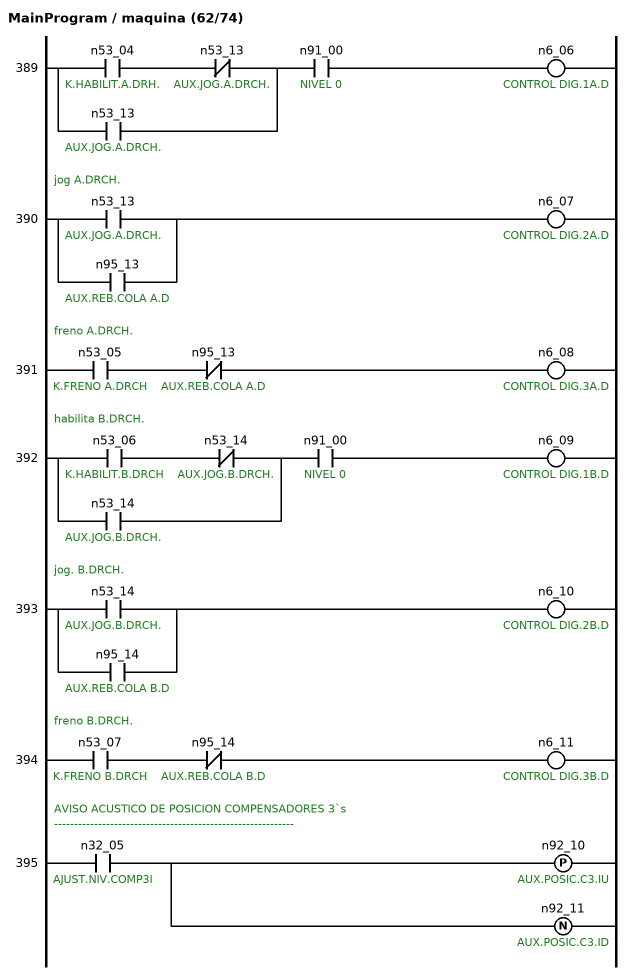
; rung 389
LD n53_04  ; K.HABILIT.A.DRH.
ANDNOT n53_13  ; AUX.JOG.A.DRCH.
OR n53_13  ; AUX.JOG.A.DRCH.
AND n91_00  ; NIVEL 0
OUT n6_06  ; CONTROL DIG.1A.D
; rung 390: jog A.DRCH.
LD n53_13  ; AUX.JOG.A.DRCH.
OR n95_13  ; AUX.REB.COLA A.D
OUT n6_07  ; CONTROL DIG.2A.D
; rung 391: freno A.DRCH.
LD n53_05  ; K.FRENO A.DRCH
ANDNOT n95_13  ; AUX.REB.COLA A.D
OUT n6_08  ; CONTROL DIG.3A.D
; rung 392: habilita B.DRCH.
LD n53_06  ; K.HABILIT.B.DRCH
ANDNOT n53_14  ; AUX.JOG.B.DRCH.
OR n53_14  ; AUX.JOG.B.DRCH.
AND n91_00  ; NIVEL 0
OUT n6_09  ; CONTROL DIG.1B.D
; rung 393: jog. B.DRCH.
LD n53_14  ; AUX.JOG.B.DRCH.
OR n95_14  ; AUX.REB.COLA B.D
OUT n6_10  ; CONTROL DIG.2B.D
; rung 394: freno B.DRCH.
LD n53_07  ; K.FRENO B.DRCH
ANDNOT n95_14  ; AUX.REB.COLA B.D
OUT n6_11  ; CONTROL DIG.3B.D
; rung 395: AVISO ACUSTICO DE POSICION COMPENSADORES 3`s / ------------------------------------------------------------
LD n32_05  ; AJUST.NIV.COMP3I
DIFU(013) n92_10  ; AUX.POSIC.C3.IU
DIFD(014) n92_11  ; AUX.POSIC.C3.ID

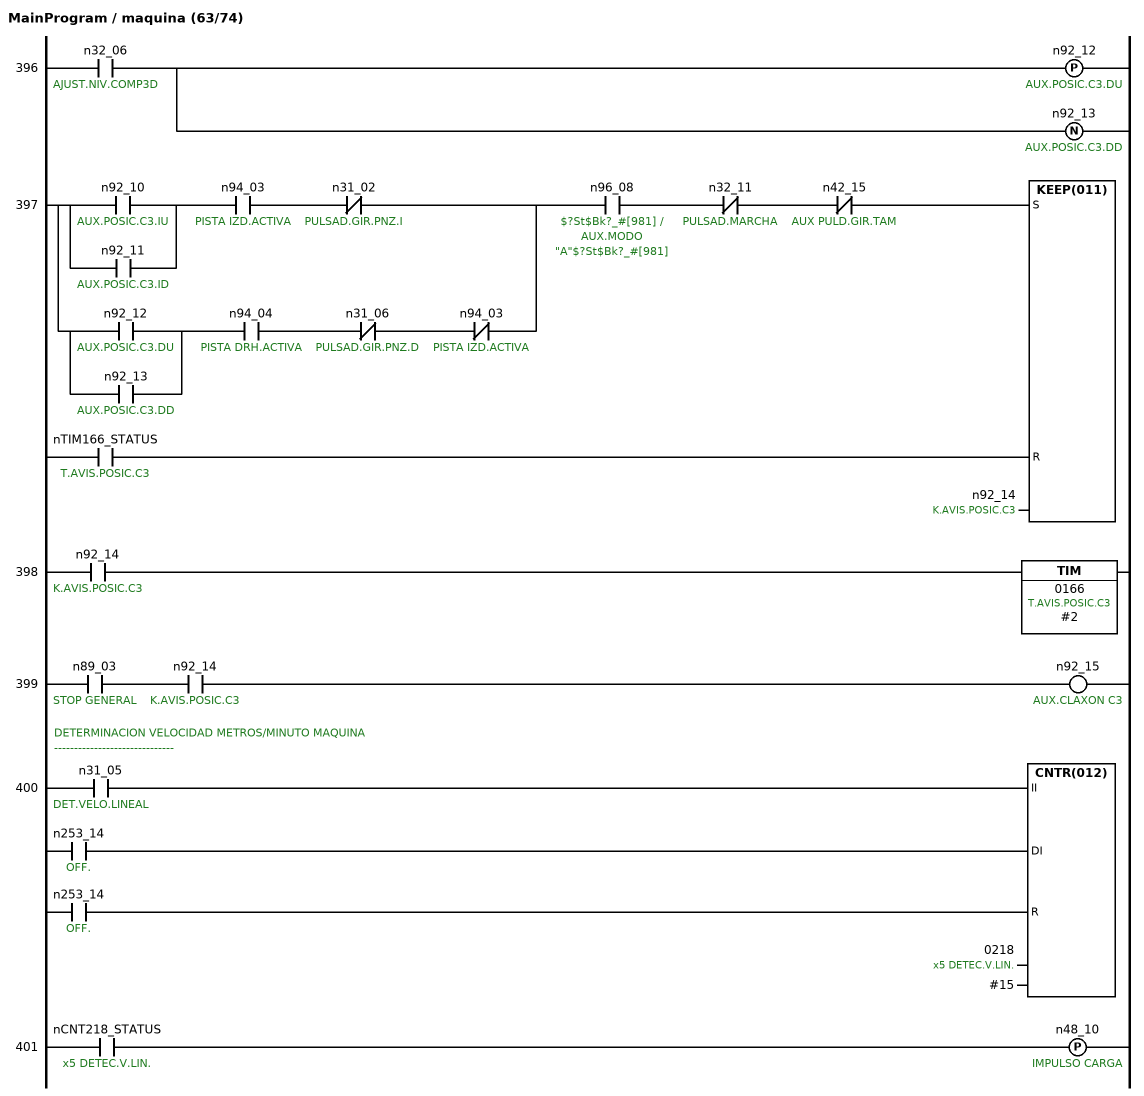
; rung 396
LD n32_06  ; AJUST.NIV.COMP3D
DIFU(013) n92_12  ; AUX.POSIC.C3.DU
DIFD(014) n92_13  ; AUX.POSIC.C3.DD
; rung 397
LD n92_10  ; AUX.POSIC.C3.IU
OR n92_11  ; AUX.POSIC.C3.ID
AND n94_03  ; PISTA IZD.ACTIVA
ANDNOT n31_02  ; PULSAD.GIR.PNZ.I
LD n92_12  ; AUX.POSIC.C3.DU
OR n92_13  ; AUX.POSIC.C3.DD
AND n94_04  ; PISTA DRH.ACTIVA
ANDNOT n31_06  ; PULSAD.GIR.PNZ.D
ANDNOT n94_03  ; PISTA IZD.ACTIVA
ORLD
AND n96_08  ; $?St$Bk?_#[981] / AUX.MODO "A"$?St$Bk?_#[981]
ANDNOT n32_11  ; PULSAD.MARCHA
ANDNOT n42_15  ; AUX PULD.GIR.TAM
LD nTIM166_STATUS  ; T.AVIS.POSIC.C3
KEEP(011) n92_14  ; K.AVIS.POSIC.C3
; rung 398
LD n92_14  ; K.AVIS.POSIC.C3
TIM 0166 #2  ; T.AVIS.POSIC.C3
; rung 399
LD n89_03  ; STOP GENERAL
AND n92_14  ; K.AVIS.POSIC.C3
OUT n92_15  ; AUX.CLAXON C3
; rung 400: DETERMINACION VELOCIDAD METROS/MINUTO MAQUINA / ------------------------------ /  / 
LD n31_05  ; DET.VELO.LINEAL
LD n253_14  ; OFF.
LD n253_14  ; OFF.
CNTR(012) 0218 #15  ; x5 DETEC.V.LIN.
; rung 401
LD nCNT218_STATUS  ; x5 DETEC.V.LIN.
DIFU(013) n48_10  ; IMPULSO CARGA

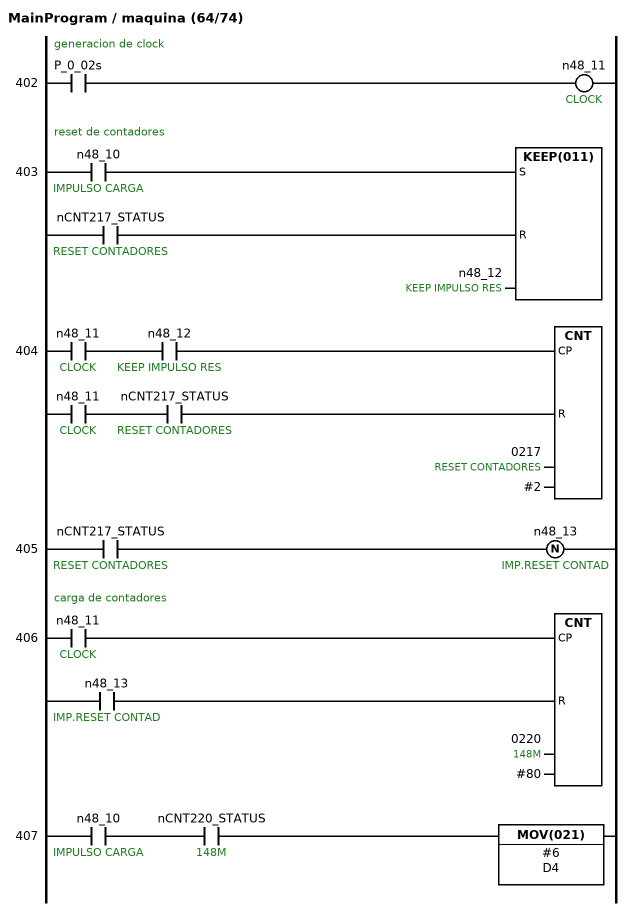
; rung 402: generacion de clock
LD P_0_02s
OUT n48_11  ; CLOCK
; rung 403: reset de contadores
LD n48_10  ; IMPULSO CARGA
LD nCNT217_STATUS  ; RESET CONTADORES
KEEP(011) n48_12  ; KEEP IMPULSO RES
; rung 404
LD n48_11  ; CLOCK
AND n48_12  ; KEEP IMPULSO RES
LD n48_11  ; CLOCK
AND nCNT217_STATUS  ; RESET CONTADORES
CNT 0217 #2  ; RESET CONTADORES
; rung 405
LD nCNT217_STATUS  ; RESET CONTADORES
DIFD(014) n48_13  ; IMP.RESET CONTAD
; rung 406: carga de contadores
LD n48_11  ; CLOCK
LD n48_13  ; IMP.RESET CONTAD
CNT 0220 #80  ; 148M
; rung 407
LD n48_10  ; IMPULSO CARGA
AND nCNT220_STATUS  ; 148M
MOV(021) #6 D4

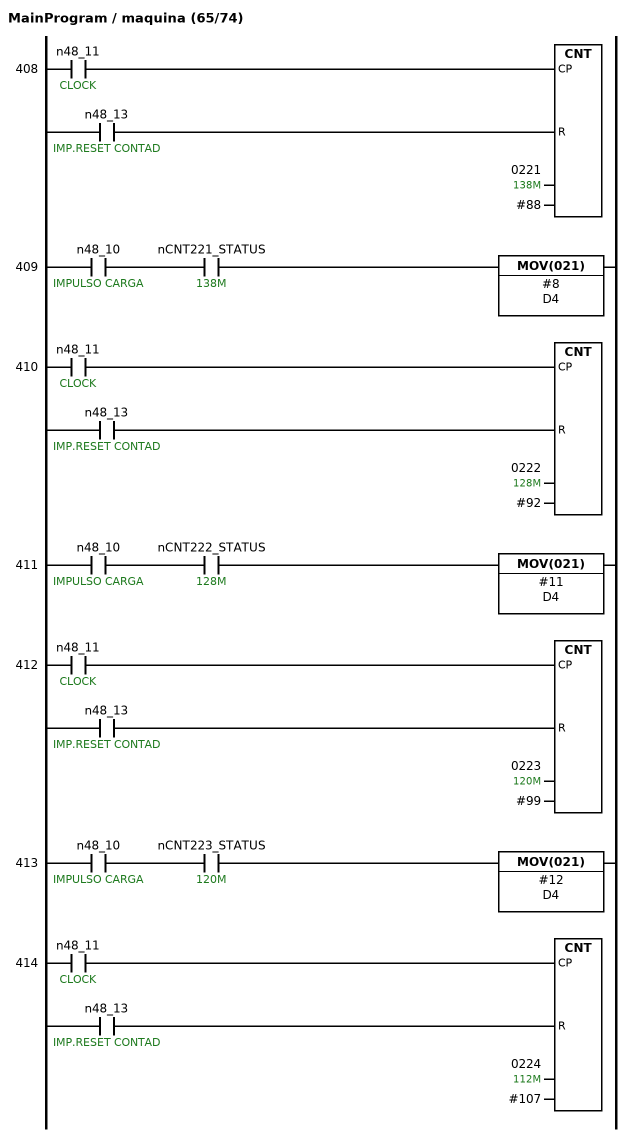
; rung 408
LD n48_11  ; CLOCK
LD n48_13  ; IMP.RESET CONTAD
CNT 0221 #88  ; 138M
; rung 409
LD n48_10  ; IMPULSO CARGA
AND nCNT221_STATUS  ; 138M
MOV(021) #8 D4
; rung 410
LD n48_11  ; CLOCK
LD n48_13  ; IMP.RESET CONTAD
CNT 0222 #92  ; 128M
; rung 411
LD n48_10  ; IMPULSO CARGA
AND nCNT222_STATUS  ; 128M
MOV(021) #11 D4
; rung 412
LD n48_11  ; CLOCK
LD n48_13  ; IMP.RESET CONTAD
CNT 0223 #99  ; 120M
; rung 413
LD n48_10  ; IMPULSO CARGA
AND nCNT223_STATUS  ; 120M
MOV(021) #12 D4
; rung 414
LD n48_11  ; CLOCK
LD n48_13  ; IMP.RESET CONTAD
CNT 0224 #107  ; 112M

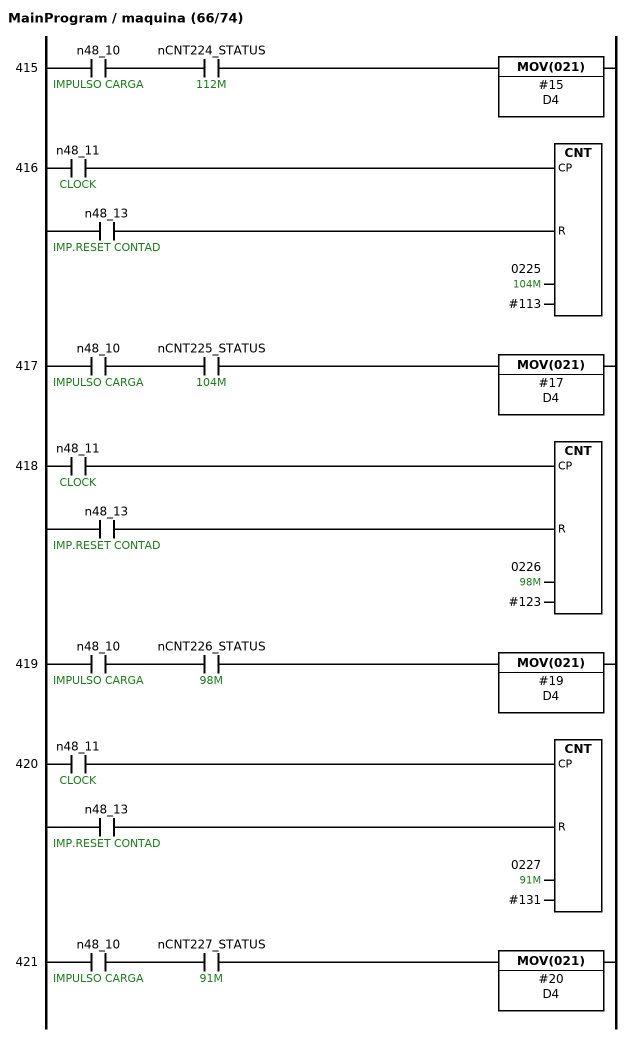
; rung 415
LD n48_10  ; IMPULSO CARGA
AND nCNT224_STATUS  ; 112M
MOV(021) #15 D4
; rung 416
LD n48_11  ; CLOCK
LD n48_13  ; IMP.RESET CONTAD
CNT 0225 #113  ; 104M
; rung 417
LD n48_10  ; IMPULSO CARGA
AND nCNT225_STATUS  ; 104M
MOV(021) #17 D4
; rung 418
LD n48_11  ; CLOCK
LD n48_13  ; IMP.RESET CONTAD
CNT 0226 #123  ; 98M
; rung 419
LD n48_10  ; IMPULSO CARGA
AND nCNT226_STATUS  ; 98M
MOV(021) #19 D4
; rung 420
LD n48_11  ; CLOCK
LD n48_13  ; IMP.RESET CONTAD
CNT 0227 #131  ; 91M
; rung 421
LD n48_10  ; IMPULSO CARGA
AND nCNT227_STATUS  ; 91M
MOV(021) #20 D4

